(* IEC 61131-3 sources: ServoDriveControllerCode_Gen3SOScompressor/src/FB (part 2) *)

(* ---- FB_FaultResetHandler.st ---- *)
(* ============================================================================
   FB_FaultResetHandler - Fault Reset Validation

   Project: Gen3 SOS Compressor Servo Controller
   Controller: Yaskawa MP2600iec

   Description:
   Validates fault reset conditions from the master controller.
   Pure combinational check - no state machine, no timers.

   Fault reset is valid when ALL conditions are met (level-based):
   - FaultReset is HIGH (level, not edge)
   - MotionEnable is LOW
   - System is in a fault state
   - Active fault code is not FAULT_NONE
   - DI0-DI2 bits are stable (no change from previous scan)
   - Master has mirrored the fault code on DI0-2 (MasterFaultCode matches ActiveFaultCode)

   NOTE: All inputs should be pre-filtered/debounced by the caller.

   Variables (define in MWiec GUI):
     VAR_INPUT:
       Enable           : BOOL             (* Enable fault reset handler
       FaultReset       : BOOL             (* Filtered fault reset signal from master
       MotionEnable     : BOOL             (* Filtered motion enable signal
       InFaultState     : BOOL             (* TRUE when system is in a fault state
       BitsStable       : BOOL             (* DI0-DI2 bits stable (no change from previous scan)
       ActiveFaultCode  : E_FaultCode      (* Active fault code for mirroring check
       MasterFaultCode  : E_FaultCode      (* Fault acknowledgement decoded from DI0-DI2
     VAR_OUTPUT:
       FaultResetValid  : BOOL             (* TRUE when all fault reset conditions met
   ============================================================================ *)

(* ============================================================================
   Main Logic
   ============================================================================ *)

IF NOT Enable THEN
    FaultResetValid := FALSE;
    RETURN;
END_IF;

(* Fault reset is valid when ALL conditions are met (level-based):
   - FaultReset is HIGH (level, not edge)
   - MotionEnable is LOW
   - We are in fault state
   - Active fault code is not FAULT_NONE
   - DI0-DI2 bits are stable
   - Master has mirrored the fault code on DI0-2 *)
FaultResetValid := FaultReset AND
                   (NOT MotionEnable) AND
                   InFaultState AND
                   (ActiveFaultCode <> FAULT_NONE) AND
                   BitsStable AND
                   (MasterFaultCode = ActiveFaultCode);

(* ---- FB_FaultToInt.st ---- *)
(* ============================================================================
   FB_FaultToInt - Convert Fault Code to Integer

   Project: Gen3 SOS Compressor Servo Controller
   Controller: Yaskawa MP2600iec

   Description:
   Converts an E_FaultCode enumeration value to its integer
   representation (0-7) for bit encoding operations.

   NOTE: Implemented as an FB (not an FN) to work around a MotionWorks IEC
   native-code-gen defect on FUNCTIONs with user-enum parameters.

   Variables (define in MWiec GUI):
     VAR_INPUT:
       Fault           : E_FaultCode      (* Fault code to convert
     VAR_OUTPUT:
       Value           : INT              (* Integer representation 0-7
   ============================================================================ *)

IF Fault = E_FaultCode#FAULT_NONE THEN
    Value := 0;
ELSIF Fault = E_FaultCode#FAULT_HANDSHAKE THEN
    Value := 1;
ELSIF Fault = E_FaultCode#FAULT_DRIVE THEN
    Value := 2;
ELSIF Fault = E_FaultCode#FAULT_POSITION THEN
    Value := 3;
ELSIF Fault = E_FaultCode#FAULT_HOMING_REQ THEN
    Value := 4;
ELSIF Fault = E_FaultCode#FAULT_PISTON_EXIT THEN
    Value := 5;
ELSIF Fault = E_FaultCode#FAULT_LIMIT_SWITCH THEN
    Value := 6;
ELSIF Fault = E_FaultCode#FAULT_ENCODER THEN
    Value := 7;
ELSE
    Value := 0;
END_IF;

(* ---- FB_ModeToInt.st ---- *)
(* ============================================================================
   FB_ModeToInt - Convert Operating Mode to Integer

   Project: Gen3 SOS Compressor Servo Controller
   Controller: Yaskawa MP2600iec

   Description:
   Converts an E_OperatingMode enumeration value to its integer
   representation (0-7) for bit encoding operations.

   NOTE: Implemented as an FB (not an FN) to work around a MotionWorks IEC
   native-code-gen defect on FUNCTIONs with user-enum parameters.

   Variables (define in MWiec GUI):
     VAR_INPUT:
       Mode            : E_OperatingMode  (* Operating mode to convert
     VAR_OUTPUT:
       Value           : INT              (* Integer representation 0-7
   ============================================================================ *)

IF Mode = E_OperatingMode#MODE_IDLE THEN
    Value := 0;
ELSIF Mode = E_OperatingMode#MODE_BRAKE_HOLD THEN
    Value := 1;
ELSIF Mode = E_OperatingMode#MODE_POSITION THEN
    Value := 2;
ELSIF Mode = E_OperatingMode#MODE_VELOCITY THEN
    Value := 3;
ELSIF Mode = E_OperatingMode#MODE_TORQUE THEN
    Value := 4;
ELSIF Mode = E_OperatingMode#MODE_GO_HOME THEN
    Value := 5;
ELSIF Mode = E_OperatingMode#MODE_HOME_LIMIT THEN
    Value := 6;
ELSIF Mode = E_OperatingMode#MODE_RESERVED_111 THEN
    Value := 7;
ELSE
    Value := 0;
END_IF;
